{attribute 'qualified_only'}
{attribute 'strict'}
TYPE E_SensorBrands :
(
	Sick,
	Pilz,
	Parker,
	Bosch 
);
END_TYPE

(* stored: Version 1.1.0.1, ProductVersion 3.1.4024.12
   DUT E_SensorBrands: Id {2b274c64-ae74-4a89-8e4f-177ed56e3077} *)
